DATA_BLOCK "DB_Send_FIFO"
TITLE =%version: 0.08 % CN: 20
//History:
//This version  %created_by: nlhdl %
//              %date_created: Monday, May 30, 2016 2:28:08 PM %
//              %release: VI_RAW/RA_Dev %
//
//Modification History:                                 By:      Date:     Rev:
//----------------------------------------------------  -------  --------  -----
//ra#14076: Package Instruct and report with pseudoID   nlHdL    14-06-16   0.08
//ra#9751: Add source files ECS-P to VI_RAW             nlHdL    14-12-15   0.07
//ra#9751: Add source files ECS-P to VI_RAW             nlHdL    07-12-15   0.07
//7632: Add blocks BIR12 for platform 4                 nlHdL    29-07-15   0.07
//7324: ECS-P General from the RD to RA for platform    nlHdL    06-07-15   0.06
//23859: Create and add BIR12 to the Vibes interface    nlHdL    30-04-15   0.10 ECS_BHS
//23824: Changed Record length to 202                   nlMlaut  29-04-15   0.06
//23155: TIR in message for tubtrace                    nlHdL    24-04-15   0.05
//22337: Remove the vibes1.x with the vibes 3.x         nlHdL    09-01-15   0.04
//18060: Update messages ID's for Vibes 3.2             nlHdL    01-04-14   1.10
//18032: package instr & package rep update             nlHdL    14-02-14   1.02
//Initial Version based on version 0.02 ECS-P GEN       nlHdL    07-11-13   1.01
//
FAMILY : VIBES
VERSION : 0.0


  STRUCT
   Header : "UDT_FIFO";
   Message : ARRAY  [1 .. 280 ] OF "UDT_Msg_Snd_Body";
  END_STRUCT ;
BEGIN
   Header.Status.Empty := TRUE;
   Header.Status.Prefull := FALSE;
   Header.Status.Full := FALSE;
   Header.Status.Record_Length_Too_Long := FALSE;
   Header.Status.Wrong_Record_Length := FALSE;
   Header.Status.Pointer_Out_Of_Range := FALSE;
   Header.Status.Wrong_Prefull_Value := FALSE;
   Header.Status.Blockmove_Fault := FALSE;
   Header.Setting.Prefull_Num_Of_Records := 240;
   Header.Setting.Record_Data_Length := 232;
   Header.Num_Of_Records_stored := 0;
   Header.Max_Numb_Of_Records := 0;
   Header.Next_Record_store := 0;
   Header.Next_Record_Retrieve := 0;
END_DATA_BLOCK

